//{attribute 'qualified_only'}
VAR_GLOBAL
	fbMachineState		:FB_MachineState;
	gRunningState		:RunningStatus:=RunningStatus.eManualState;
END_VAR

(* stored: Version 1.1.0.1, ProductVersion 3.1.4024.4
   GVL GVL_MachineState: Id {94a03c0c-071c-489a-94e2-2e1861c8ade1} *)
